FUNCTION_BLOCK plant
  (* Standard: 61499-2 *)
  (* Version 0.1, 2017-00-25, hpea485, UOA *)
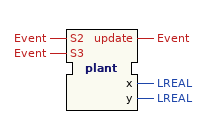
  EVENT_INPUT
    S2;
    S3;
  END_EVENT
  EVENT_OUTPUT
    update;
  END_EVENT
  VAR_OUTPUT
    x : LREAL;
    y : LREAL;
  END_VAR
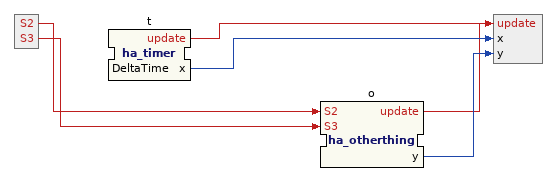
  FBS
    t : ha_timer;
    o : ha_otherthing;
  END_FBS
  EVENT_CONNECTIONS
    S2 TO o.S2;
    S3 TO o.S3;
    t.update TO update;
    o.update TO update;
  END_CONNECTIONS
  DATA_CONNECTIONS
    t.x TO x;
    o.y TO y;
  END_CONNECTIONS
END_FUNCTION_BLOCK
